{attribute 'linkalways'} 
{attribute 'no_explicit_call' := 'This FB is a CLASS and must be accessed using methods or properties'}
{attribute 'enable_dynamic_creation'}
FUNCTION_BLOCK Node_F_VN_MinElementElementwise_TcVnVector4_DINT EXTENDS VisionNode
VAR
    ipContainer : _ITcVnContainer;
    aMin : _TcVnVector4_DINT;
    hrPrev : _HRESULT(S_OK);
    hresult : _HRESULT(S_OK);
END_VAR

METHOD PUBLIC  Clone : I_Node
VAR
	pNode : POINTER TO Node_F_VN_MinElementElementwise_TcVnVector4_DINT;
END_VAR
pNode := __NEW(Node_F_VN_MinElementElementwise_TcVnVector4_DINT);
Clone := pNode^;
END_METHOD

METHOD FB_init : BOOL
VAR_INPUT
	bInitRetains : BOOL; // if TRUE, the retain variables are initialized (warm start / cold start)
	bInCopyCode : BOOL;  // if TRUE, the instance afterwards gets moved into the copy code (online change)
END_VAR
AddInput('ipContainer', ipContainer);
AddInput('hrPrev', hrPrev);
AddOutput('ipContainer', ipContainer);
AddOutput('aMin', aMin);
AddOutput('hresult',hresult);
END_METHOD

METHOD PROTECTED OnExecute
hresult.Value := F_VN_MinElementElementwise_TcVnVector4_DINT(
    ipContainer := ipContainer.Value,
    aMin := aMin.Value,
    hrPrev:= hrPrev.Value);
END_METHOD

METHOD PUBLIC PreExecutionCheck
VAR_INPUT
	Check : I_PreExecutionChecks;
END_VAR
Check.IsTrue(ipContainer.IsValid, 'ipContainer must be a valid container');
Check.IsTrue(ipContainer.IsType(TC_GLOBAL_CONST_LIST.ContainerType_Vector_TcVnVector4_DINT), 'ipContainer contains incorrect type');
END_METHOD

END_FUNCTION_BLOCK

(* stored: Version 1.1.0.1, ProductVersion 3.1.4026.13
   POU Node_F_VN_MinElementElementwise_TcVnVector4_DINT: Id {74a027a2-7eff-4aab-a65f-e941a17bd66e}, SpecialFunc None
   Folder Constructor: Id {02eceb4e-2a65-4b13-9f6a-3cb3f227b0b3}
   Method Clone: Id {324dfff1-4483-442e-95f6-2a65592eec1a}
   Method FB_init: Id {8868e50c-3d00-4e77-a354-1f4dae5fa009}
   Method OnExecute: Id {d250539d-4c83-488f-8ad0-8c00f467ab50}
   Method PreExecutionCheck: Id {336a2aee-97c4-463b-92c7-66ae7b8cfaeb} *)
